(* IEC 61131-3 sources: SRCI/RobotLibrary/Library/POUs/BasicMove/MC_ReturnToPrimary, 1 file *)

(* ---- MC_ReturnToPrimaryFB.st ---- *)
/// Return to path left during active interrupt
FUNCTION_BLOCK MC_ReturnToPrimaryFB EXTENDS RobotLibraryBaseFB
// -------------------------------------------------------------------------
//  SRCI Robot Library
// -------------------------------------------------------------------------
//
//  Object:      ReturnToPrimaryFB
//  Author:      Thorsten Brach
//  Date:        2024-06-01
//
//  Description:
//
//
//  Copyright:
//    (C) 2024 Thorsten Brach. All rights reserved
//             Licensed under the LGPL-3.0 license.
//
//  Disclaimer:
//    This project is provided without any guarantee and can be used for
//    private and commercial purposes. Any use is at the user’s
//    own risk and responsibility.
//
// -------------------------------------------------------------------------
VAR_INPUT
  /// Activate ReturnToPrimary
  Enable             : BOOL;
  /// command parameter
  ParCmd             : ReturnToPrimaryParCmd;
END_VAR

VAR_OUTPUT
  /// The command has been completed successfully
  Done               : BOOL;
  /// FB is being processed
  Busy               : BOOL;
  /// Command is transferred and confirmed by the RC
  CommandBuffered    : BOOL;
  /// The command takes control of the motion of the according axis group
  Active             : BOOL;
  /// The command was aborted by another command.
  CommandAborted     : BOOL;
  /// TRUE, while command is interrupted during execution and can be continued
  CommandInterrupted : BOOL;
  /// command results
  OutCmd             : ReturnToPrimaryOutCmd;
END_VAR

VAR
  /// internal copy of command parameter
 _parCmd             : ReturnToPrimaryParCmd;
  /// command data to send
 _command            : ReturnToPrimarySendData;
  /// response data received
 _response           : ReturnToPrimaryRecvData;
  /// Rising edge for enable
 _enable_R           : R_TRIG;
  /// Falling edge for enable
 _enable_F           : F_TRIG;
END_VAR

  SUPER^(AxesGroup := AxesGroup);

END_FUNCTION_BLOCK

METHOD INTERNAL CheckAddParameter : BOOL
VAR_INPUT
  /// Payload pointer
  PayloadPtr : UDINT;
END_VAR
VAR
  /// Payload as byte array
  Payload    : ARRAY [1..SIZEOF(_command)] OF BYTE;
  /// Null Byte array
  Null       : ARRAY [1..SIZEOF(_command)] OF BYTE;
  /// Data length to compare
  DataLen    : UDINT;
END_VAR

  // Payload pointer must be decreased by one byte, because ADR(Payload) is already one byte !
  PayloadPtr := LIMIT (0, PayloadPtr - 1, SIZEOF(Payload) -1);
  // Convert command struct to payload array
  SysDepMemCpy( pDest := ADR(Payload), pSrc := ADR(_command), DataLen := SIZEOF(_command));
  // Calculate the data length to compare - at least one byte must be compared !
  DataLen := LIMIT(1, SIZEOF(Payload) - PayloadPtr, SIZEOF(Payload));
  // Compare Payload-Array with Null-Byte-Array
  CheckAddParameter := SysDepMemCmp( pData1 := ADR(Payload) + PayloadPtr , pData2 := ADR(Null), DataLen := DataLen) <>  RobotLibraryConstants.OK ;

END_METHOD

METHOD PROTECTED CheckFunctionSupported : BOOL
VAR_IN_OUT
  /// Robot assignment of function
  AxesGroup : AxesGroup;
END_VAR

  CheckFunctionSupported := AxesGroup.State.RobotData.RCSupportedFunctions.ReturnToPrimary;

  IF ( NOT CheckFunctionSupported )
  THEN
    // call base implementation for set error and create log entry
    SUPER^.CheckFunctionSupported(AxesGroup := AxesGroup);
  END_IF

END_METHOD

METHOD PROTECTED CheckParameterChanged : BOOL
VAR_IN_OUT
  /// Robot assignment of function
  AxesGroup    : AxesGroup;
END_VAR

  // Check ParCmd Size is > 0, because MemCmp does not work correctly with size = 0
  IF (SIZEOF(ParCmd) = 0) OR (_stepCmd = 0)
  THEN
    RETURN;
  END_IF

  // compare memory
  _parameterChanged := ( SysDepMemCmp(pData1 := ADR(ParCmd), pData2 := ADR(_parCmd), DataLen := SIZEOF(ParCmd)) <> RobotLibraryConstants.OK );

  // check parameter valid ?
  _parameterValid   := CheckParameterValid( AxesGroup := AxesGroup );

  IF ((  _parameterChanged        )  AND
      (  _parameterValid          )) OR
      (  _parameterUpdateInternal )
  THEN
    // reset internal flag for send parameter update
   _parameterUpdateInternal := FALSE;
    // update internal copy of parameters
   _parCmd := ParCmd;
    // inc parameter sequence
   _command.ParSeq := _command.ParSeq + 1;
    // update command data
    CommandData := CreateCommandPayload(AxesGroup := AxesGroup); // ( Access via reference to rCommandFB in ACR )
    // notify active command register
    AxesGroup.Acyclic.ActiveCommandRegister.NotifyParameterChanged := _uniqueID;
  END_IF

END_METHOD

METHOD PROTECTED CheckParameterValid : BOOL
VAR_IN_OUT
  /// Robot assignment of function
  AxesGroup : AxesGroup;
END_VAR
VAR
  /// internal index for loops
 _idx : DINT;
END_VAR

  CheckParameterValid := TRUE;

  // Check ParCmd.ReturnMode valid ?
  IF (( ParCmd.ReturnMode <> ReturnMode.INTERRUPT_POSITION ) AND
      ( ParCmd.ReturnMode <> ReturnMode.END_POSITION       ))
  THEN
    // Parameter not valid
    CheckParameterValid := FALSE;
    // Set error
    ErrorID := RobotLibraryErrorIdEnum.ERR_INVALID_PAR_CMD;
    // Create log entry
    CreateLogMessagePara1 ( Timestamp   := AxesGroup.State.SystemTime,
                            MessageType := MessageType.CMD,
                            Severity    := Severity.ERROR,
                            MessageCode := ErrorID,
                            MessageText := 'Invalid Parameter ParCmd.ReturnMode = {1}',
                            Para1       := RETURN_MODE_TO_STRING(ParCmd.ReturnMode));
    RETURN;
  END_IF

  // Check ParCmd.VelocityRate valid ?
  IF  (( SysDepIsValidReal(ParCmd.VelocityRate) = FALSE )  OR
      ((                   ParCmd.VelocityRate  <     0 )  AND
       (                   ParCmd.VelocityRate <>    -1 )) OR
       (                   ParCmd.VelocityRate  >   100 ))
  THEN
    // Parameter not valid
    CheckParameterValid := FALSE;
    // Set error
    ErrorID := RobotLibraryErrorIdEnum.ERR_VELOCITY_INVALID;
    // Create log entry
    CreateLogMessagePara1 ( Timestamp   := AxesGroup.State.SystemTime,
                            MessageType := MessageType.CMD,
                            Severity    := Severity.ERROR,
                            MessageCode := ErrorID,
                            MessageText := 'Invalid Parameter ParCmd.VelocityRate = {1}',
                            Para1       := VALID_REAL_TO_STRING(ParCmd.VelocityRate));
    RETURN;
  END_IF

  // Check ParCmd.AccelerationRate valid ?
  IF  (( SysDepIsValidReal(ParCmd.AccelerationRate) = FALSE )  OR
      ((                   ParCmd.AccelerationRate  <     0 )  AND
       (                   ParCmd.AccelerationRate <>    -1 )) OR
       (                   ParCmd.AccelerationRate  >   100 ))
  THEN
    // Parameter not valid
    CheckParameterValid := FALSE;
    // Set error
    ErrorID := RobotLibraryErrorIdEnum.ERR_ACCELERATION_INVALID;
    // Create log entry
    CreateLogMessagePara1 ( Timestamp   := AxesGroup.State.SystemTime,
                            MessageType := MessageType.CMD,
                            Severity    := Severity.ERROR,
                            MessageCode := ErrorID,
                            MessageText := 'Invalid Parameter ParCmd.AccelerationRate = {1}',
                            Para1       := VALID_REAL_TO_STRING(ParCmd.AccelerationRate));
    RETURN;
  END_IF

  // Check ParCmd.DecelerationRate valid ?
  IF  (( SysDepIsValidReal(ParCmd.DecelerationRate) = FALSE )  OR
      ((                   ParCmd.DecelerationRate  <     0 )  AND
       (                   ParCmd.DecelerationRate <>    -1 )) OR
       (                   ParCmd.DecelerationRate  >   100 ))
  THEN
    // Parameter not valid
    CheckParameterValid := FALSE;
    // Set error
    ErrorID := RobotLibraryErrorIdEnum.ERR_DECELERATION_INVALID;
    // Create log entry
    CreateLogMessagePara1 ( Timestamp   := AxesGroup.State.SystemTime,
                            MessageType := MessageType.CMD,
                            Severity    := Severity.ERROR,
                            MessageCode := ErrorID,
                            MessageText := 'Invalid Parameter ParCmd.DecelerationRate = {1}',
                            Para1       := VALID_REAL_TO_STRING(ParCmd.DecelerationRate));
    RETURN;
  END_IF

  // Check ParCmd.JerkRate valid ?
  IF  (( SysDepIsValidReal(ParCmd.JerkRate) = FALSE )  OR
      ((                   ParCmd.JerkRate  <     0 )  AND
       (                   ParCmd.JerkRate <>    -1 )) OR
       (                   ParCmd.JerkRate  >   100 ))
  THEN
    // Parameter not valid
    CheckParameterValid := FALSE;
    // Set error
    ErrorID := RobotLibraryErrorIdEnum.ERR_JERK_INVALID;
    // Create log entry
    CreateLogMessagePara1 ( Timestamp   := AxesGroup.State.SystemTime,
                            MessageType := MessageType.CMD,
                            Severity    := Severity.ERROR,
                            MessageCode := ErrorID,
                            MessageText := 'Invalid Parameter ParCmd.JerkRate = {1}',
                            Para1       := VALID_REAL_TO_STRING(ParCmd.JerkRate));
    RETURN;
  END_IF

  // Check ParCmd.ToolNo valid ?
  IF (( ParCmd.ToolNo <   0                                                ) OR
      ( ParCmd.ToolNo > 254                                                ) OR
      ( ParCmd.ToolNo > AxesGroup.State.ConfigurationData.HighestToolIndex ) OR
      ( ParCmd.ToolNo > RobotLibraryParameter.TOOL_MAX -1                  ))
  THEN
    // Parameter not valid
    CheckParameterValid := FALSE;

    // Check ToolNo available on RC ?
    IF ( ParCmd.ToolNo > AxesGroup.State.ConfigurationData.HighestToolIndex )
    THEN
      ErrorID := RobotLibraryErrorIdEnum.ERR_TOOLNO_UNAVAILABLE;
    ELSE
      ErrorID := RobotLibraryErrorIdEnum.ERR_TOOLNO_RANGE;
  	END_IF

    // Create log entry
    CreateLogMessagePara1 ( Timestamp   := AxesGroup.State.SystemTime,
                            MessageType := MessageType.CMD,
                            Severity    := Severity.ERROR,
                            MessageCode := ErrorID,
                            MessageText := 'Invalid Parameter ParCmd.ToolNo = {1}',
                            Para1       := USINT_TO_STRING(ParCmd.ToolNo));
    RETURN;
  END_IF

  // Check ParCmd.FrameNo valid ?
  IF (( ParCmd.FrameNo <   0                                                 ) OR
      ( ParCmd.FrameNo > 254                                                 ) OR
      ( ParCmd.FrameNo > AxesGroup.State.ConfigurationData.HighestFrameIndex ) OR
      ( ParCmd.FrameNo > RobotLibraryParameter.FRAME_MAX -1                  ))
  THEN
    // Parameter not valid
    CheckParameterValid := FALSE;

    // Check FrameNo available on RC ?
    IF ( ParCmd.FrameNo > AxesGroup.State.ConfigurationData.HighestFrameIndex )
    THEN
      ErrorID := RobotLibraryErrorIdEnum.ERR_FRAMENO_UNAVAILABLE;
    ELSE
      ErrorID := RobotLibraryErrorIdEnum.ERR_FRAMENO_RANGE;
  	END_IF

    // Create log entry
    CreateLogMessagePara1 ( Timestamp   := AxesGroup.State.SystemTime,
                            MessageType := MessageType.CMD,
                            Severity    := Severity.ERROR,
                            MessageCode := ErrorID,
                            MessageText := 'Invalid Parameter ParCmd.FrameNo = {1}',
                            Para1       := USINT_TO_STRING(ParCmd.FrameNo));
    RETURN;
  END_IF

  // Check ParCmd.DistanceLimit valid ?
  IF  ( SysDepIsValidReal(ParCmd.DistanceLimit) = FALSE )
  THEN
    // Parameter not valid
    CheckParameterValid := FALSE;
    // Set error
    ErrorID := RobotLibraryErrorIdEnum.ERR_JERK_INVALID;
    // Create log entry
    CreateLogMessagePara1 ( Timestamp   := AxesGroup.State.SystemTime,
                            MessageType := MessageType.CMD,
                            Severity    := Severity.ERROR,
                            MessageCode := ErrorID,
                            MessageText := 'Invalid Parameter ParCmd.DistanceLimit = {1}',
                            Para1       := VALID_REAL_TO_STRING(ParCmd.DistanceLimit));
    RETURN;
  END_IF

  // Check ParCmd.TrajectoryMode valid ?
  IF (( ParCmd.TrajectoryMode <> TrajectoryMode.INVALID         ) AND
      ( ParCmd.TrajectoryMode <> TrajectoryMode.LINEAR_MOVEMENT ) AND
      ( ParCmd.TrajectoryMode <> TrajectoryMode.PTP_MOVEMENT    ))
  THEN
    // Parameter not valid
    CheckParameterValid := FALSE;
    // Set error
    ErrorID := RobotLibraryErrorIdEnum.ERR_TRAJECTORYMODE_INVALID;
    // Create log entry
    CreateLogMessagePara1 ( Timestamp   := AxesGroup.State.SystemTime,
                            MessageType := MessageType.CMD,
                            Severity    := Severity.ERROR,
                            MessageCode := ErrorID,
                            MessageText := 'Invalid Parameter ParCmd.TrajectoryMode = {1}',
                            Para1       := TRAJECTORY_MODE_TO_STRING(ParCmd.TrajectoryMode));
    RETURN;
  END_IF

  // Check ParCmd.MoveTime valid ?
  IF  ( ParCmd.MoveTime < T#0S )
  THEN
    // Parameter not valid
    CheckParameterValid := FALSE;
    // Set error
    ErrorID := RobotLibraryErrorIdEnum.ERR_INVALID_PAR_CMD;
    // Create log entry
    CreateLogMessagePara1 ( Timestamp   := AxesGroup.State.SystemTime,
                            MessageType := MessageType.CMD,
                            Severity    := Severity.ERROR,
                            MessageCode := ErrorID,
                            MessageText := 'Invalid Parameter ParCmd.MoveTime = {1}',
                            Para1       := TIME_TO_STRING(ParCmd.MoveTime));
    RETURN;
  END_IF

  // Check ParCmd.AllowDifferences
  // -> no plausibility check for boolean

END_METHOD

METHOD INTERNAL CreateCommandPayload : RobotLibraryCommandDataFB
VAR_IN_OUT
  /// Robot assignment of function
  AxesGroup : AxesGroup;
END_VAR
VAR
  /// Parameter count
 _parameterCnt : DINT;
END_VAR
// Table 6-310: Sent CMD payload (PLC to RC) of "ReturnToPrimary"
// --------------------------
// Header
// --------------------------
// Byte 00 : UINT  - Type HB
// Byte 01 :       - Type LB
// Byte 02 : USINT - Reserve | ExecutionMode
// Byte 03 : USINT - ParSeq  | Priority
// --------------------------
// Datablock
// --------------------------
// Byte 04  : UINT  - VelocityRate LW HB
// Byte 05  :       - VelocityRate LW LB
// Byte 06  : UINT  - AccelerationRate LW HB
// Byte 07  :       - AccelerationRate LW LB
// Byte 08  : UINT  - DecelerationRate LW HB
// Byte 09  :       - DecelerationRate LW LB
// Byte 10  : UINT  - JerkRate LW HB
// Byte 11  :       - JerkRate LW LB
// Byte 12  : REAL  - DistanceLimit HW HB
// Byte 13  :       - DistanceLimit HW LB
// Byte 14  :       - DistanceLimit LW HB
// Byte 15  :       - DistanceLimit LW LB
// Byte 16  : USINT - ToolNo
// Byte 17  : USINT - FrameNo
// Byte 18  : UINT  - Move Time LW HB
// Byte 19  : UINT  - Move Time LW LB
// Byte 20  : BYTE  - BIT 00 : ReturnMode
//                    BIT 01 : TrajectoryMode
//                    BIT 02 : Enable
//                    BIT 03 : AllowDifferences
// Byte 21  : BYTE  - PaddingByte

// --------------------------
VAR
 _tmpByte : BYTE;
END_VAR

  // set command parameter
  _command.CmdTyp            :=  CmdType.ReturnToPrimary;
  _command.ExecMode          :=  ExecMode;
  _command.ParSeq            := _command.ParSeq;
  _command.Priority          :=  Priority;
  _command.ToolNo            := _parCmd.ToolNo;
  _command.FrameNo           := _parCmd.FrameNo;
  _command.VelocityRate      :=  REAL_TO_PERCENT_UINT(_parCmd.VelocityRate     , IsOptional := FALSE);
  _command.AccelerationRate  :=  REAL_TO_PERCENT_UINT(_parCmd.AccelerationRate , IsOptional := FALSE);
  _command.DecelerationRate  :=  REAL_TO_PERCENT_UINT(_parCmd.DecelerationRate , IsOptional := TRUE );
  _command.JerkRate          :=  REAL_TO_PERCENT_UINT(_parCmd.JerkRate         , IsOptional := TRUE );
  _command.DistanceLimit     := _parCmd.DistanceLimit;
  _command.ReturnMode        :=(_parCmd.ReturnMode = ReturnMode.END_POSITION);
  _command.TrajectoryMode    := _parCmd.TrajectoryMode = TrajectoryMode.PTP_MOVEMENT;
  _command.MoveTime          :=  TIME_TO_UINT(_parCmd.MoveTime);
  _command.Enable            :=  Enable;

  // copy command data to header
  _cmdHeader := _command;
  // call base implementation to copy header to payload buffer
  CreateCommandPayload := SUPER^.CreateCommandPayload(AxesGroup := AxesGroup);

  {warning 'ToDo: Changes in Spec V1.5, which are different to Spec V1.3'}

  // Check parameter must be added ?
  IF ( CheckAddParameter(CreateCommandPayload.PayloadPtr))
  THEN
    // add command.VelocityRate
    CreateCommandPayload.AddUint(_command.VelocityRate);
    // inc parameter counter
   _parameterCnt := _parameterCnt + 1;
  END_IF

  // Check parameter must be added ?
  IF ( CheckAddParameter(CreateCommandPayload.PayloadPtr))
  THEN
    // add command.AccelerationRate
    CreateCommandPayload.AddUint(_command.AccelerationRate);
    // inc parameter counter
   _parameterCnt := _parameterCnt + 1;
  END_IF

  // Check parameter must be added ?
  IF ( CheckAddParameter(CreateCommandPayload.PayloadPtr))
  THEN
    // add command.DecelerationRate
    CreateCommandPayload.AddUint(_command.DecelerationRate);
    // inc parameter counter
   _parameterCnt := _parameterCnt + 1;
  END_IF

  // Check parameter must be added ?
  IF ( CheckAddParameter(CreateCommandPayload.PayloadPtr))
  THEN
    // add command.JerkRate
    CreateCommandPayload.AddUint(_command.JerkRate);
    // inc parameter counter
   _parameterCnt := _parameterCnt + 1;
  END_IF

  // Check parameter must be added ?
  IF ( CheckAddParameter(CreateCommandPayload.PayloadPtr))
  THEN
    // add command.DistanceLimit
    CreateCommandPayload.AddReal(_command.DistanceLimit);
    // inc parameter counter
   _parameterCnt := _parameterCnt + 1;
  END_IF

  // Check parameter must be added ?
  IF ( CheckAddParameter(CreateCommandPayload.PayloadPtr))
  THEN
    // add command.ToolNo
    CreateCommandPayload.AddUsint(_command.ToolNo);
    // inc parameter counter
   _parameterCnt := _parameterCnt + 1;
  END_IF

  // Check parameter must be added ?
  IF ( CheckAddParameter(CreateCommandPayload.PayloadPtr))
  THEN
    // add command.FrameNo
    CreateCommandPayload.AddUsint(_command.FrameNo);
    // inc parameter counter
   _parameterCnt := _parameterCnt + 1;
  END_IF

  // Check parameter must be added ?
  IF ( CheckAddParameter(CreateCommandPayload.PayloadPtr))
  THEN
    // add command.MoveTime
    CreateCommandPayload.AddUint(_command.MoveTime);
    // inc parameter counter
   _parameterCnt := _parameterCnt + 1;
  END_IF

  // Check parameter must be added ?
  IF ( CheckAddParameter(CreateCommandPayload.PayloadPtr))
  THEN
   _tmpByte.0 := _command.ReturnMode;
   _tmpByte.1 := _command.TrajectoryMode;
   _tmpByte.2 := _command.Enable;
   _tmpByte.3 := _command.AllowDifferences;
    // add command.ReturnMode
    CreateCommandPayload.AddByte(_tmpByte);
    // inc parameter counter
   _parameterCnt := _parameterCnt + 1;
  END_IF

  // Create logging
  CreateCommandPayloadLog(AxesGroup := AxesGroup, ParameterCnt := _parameterCnt);

END_METHOD

METHOD INTERNAL CreateCommandPayloadLog
VAR_IN_OUT
  /// Robot assignment of function
  AxesGroup : AxesGroup;
END_VAR
VAR_INPUT
  /// Parameter count
  ParameterCnt : DINT;
END_VAR

  // Create log entry for Parameter start
  CreateLogMessagePara1 ( Timestamp   := AxesGroup.State.SystemTime,
                          MessageType := MessageType.CMD,
                          Severity    := Severity.DEBUG,
                          MessageCode := 0,
                          MessageText := 'Create command payload with the {1} parameter(s) :',
                          Para1       := DINT_TO_STRING(ParameterCnt));

  // Return if no parameter is remaining...
  IF ( ParameterCnt = 0 ) THEN RETURN; END_IF
  // dec remaining parameter(s)
  ParameterCnt := ParameterCnt - 1;
  // Create log entry for ToolNo
  CreateLogMessagePara1 ( Timestamp   := AxesGroup.State.SystemTime,
                          MessageType := MessageType.CMD,
                          Severity    := Severity.DEBUG,
                          MessageCode := 0,
                          MessageText := 'Command.ToolNo = {1}',
                          Para1       :=  USINT_TO_STRING(_command.ToolNo));

  // Return if no parameter is remaining...
  IF ( ParameterCnt = 0 ) THEN RETURN; END_IF
  // dec remaining parameter(s)
  ParameterCnt := ParameterCnt - 1;
  // Create log entry for FrameNo
  CreateLogMessagePara1 ( Timestamp   := AxesGroup.State.SystemTime,
                          MessageType := MessageType.CMD,
                          Severity    := Severity.DEBUG,
                          MessageCode := 0,
                          MessageText := 'Command.FrameNo = {1}',
                          Para1       :=  USINT_TO_STRING(_command.FrameNo));

  // Return if no parameter is remaining...
  IF ( ParameterCnt = 0 ) THEN RETURN; END_IF
  // dec remaining parameter(s)
  ParameterCnt := ParameterCnt - 1;
  // Create log entry for VelocityRate
  CreateLogMessagePara1 ( Timestamp   := AxesGroup.State.SystemTime,
                          MessageType := MessageType.CMD,
                          Severity    := Severity.DEBUG,
                          MessageCode := 0,
                          MessageText := 'Command.VelocityRate = {1}',
                          Para1       :=  UINT_TO_STRING(_command.VelocityRate));

  // Return if no parameter is remaining...
  IF ( ParameterCnt = 0 ) THEN RETURN; END_IF
  // dec remaining parameter(s)
  ParameterCnt := ParameterCnt - 1;
  // Create log entry for AccelerationRate
  CreateLogMessagePara1 ( Timestamp   := AxesGroup.State.SystemTime,
                          MessageType := MessageType.CMD,
                          Severity    := Severity.DEBUG,
                          MessageCode := 0,
                          MessageText := 'Command.AccelerationRate = {1}',
                          Para1       :=  UINT_TO_STRING(_command.AccelerationRate));

  // Return if no parameter is remaining...
  IF ( ParameterCnt = 0 ) THEN RETURN; END_IF
  // dec remaining parameter(s)
  ParameterCnt := ParameterCnt - 1;
  // Create log entry for DecelerationRate
  CreateLogMessagePara1 ( Timestamp   := AxesGroup.State.SystemTime,
                          MessageType := MessageType.CMD,
                          Severity    := Severity.DEBUG,
                          MessageCode := 0,
                          MessageText := 'Command.DecelerationRate = {1}',
                          Para1       :=  UINT_TO_STRING(_command.DecelerationRate));

  // Return if no parameter is remaining...
  IF ( ParameterCnt = 0 ) THEN RETURN; END_IF
  // dec remaining parameter(s)
  ParameterCnt := ParameterCnt - 1;
  // Create log entry for JerkRate
  CreateLogMessagePara1 ( Timestamp   := AxesGroup.State.SystemTime,
                          MessageType := MessageType.CMD,
                          Severity    := Severity.DEBUG,
                          MessageCode := 0,
                          MessageText := 'Command.JerkRate = {1}',
                          Para1       :=  UINT_TO_STRING(_command.JerkRate));

  // Return if no parameter is remaining...
  IF ( ParameterCnt = 0 ) THEN RETURN; END_IF
  // dec remaining parameter(s)
  ParameterCnt := ParameterCnt - 1;
  // Create log entry for DistanceLimit
  CreateLogMessagePara1 ( Timestamp   := AxesGroup.State.SystemTime,
                          MessageType := MessageType.CMD,
                          Severity    := Severity.DEBUG,
                          MessageCode := 0,
                          MessageText := 'Command.DistanceLimit = {1}',
                          Para1       :=  REAL_TO_STRING(_command.DistanceLimit));

  // Return if no parameter is remaining...
  IF ( ParameterCnt = 0 ) THEN RETURN; END_IF
  // dec remaining parameter(s)
  ParameterCnt := ParameterCnt - 1;
  // Create log entry for ReturnMode
  CreateLogMessagePara1 ( Timestamp   := AxesGroup.State.SystemTime,
                          MessageType := MessageType.CMD,
                          Severity    := Severity.DEBUG,
                          MessageCode := 0,
                          MessageText := 'Command.ReturnMode = {1}',
                          Para1       :=  BOOL_TO_STRING(_command.ReturnMode));

  // Return if no parameter is remaining...
  IF ( ParameterCnt = 0 ) THEN RETURN; END_IF
  // dec remaining parameter(s)
  ParameterCnt := ParameterCnt - 1;
  // Create log entry for TrajectoryMode
  CreateLogMessagePara1 ( Timestamp   := AxesGroup.State.SystemTime,
                          MessageType := MessageType.CMD,
                          Severity    := Severity.DEBUG,
                          MessageCode := 0,
                          MessageText := 'Command.TrajectoryMode = {1}',
                          Para1       :=  BOOL_TO_STRING(_command.TrajectoryMode));

  // Return if no parameter is remaining...
  IF ( ParameterCnt = 0 ) THEN RETURN; END_IF
  // dec remaining parameter(s)
  ParameterCnt := ParameterCnt - 1;
  // Create log entry for MoveTime
  CreateLogMessagePara1 ( Timestamp   := AxesGroup.State.SystemTime,
                          MessageType := MessageType.CMD,
                          Severity    := Severity.DEBUG,
                          MessageCode := 0,
                          MessageText := 'Command.MoveTime = {1}',
                          Para1       :=  UINT_TO_STRING(_command.MoveTime));

END_METHOD

METHOD FB_init : BOOL
VAR_INPUT
  /// if TRUE, the retain variables are initialized (warm start / cold start)
  bInitRetains : BOOL;
  /// if TRUE, the instance afterwards gets moved into the copy code (online change)
  bInCopyCode  : BOOL;
END_VAR

  MyType := 'MC_ReturnToPrimaryFB';

  ExecMode := ExecutionMode.SEQUENCE_PRIMARY;
  Priority := PriorityLevel.NORMAL;

END_METHOD

METHOD PROTECTED OnExecRun : DINT
VAR_IN_OUT
  /// Robot assignment of function
  AxesGroup : AxesGroup;
END_VAR

  // call base implementation
  SUPER^.OnExecRun(AxesGroup := AxesGroup);

  // building rising and falling edges
  _enable_R( CLK := Enable);
  _enable_F( CLK := Enable);

  CASE _stepCmd OF

    00:  IF ( _enable_R.Q ) AND ( NOT Error)
         THEN
           // reset the rising edge
          _enable_R();
           // reset the falling edge
          _enable_F();

           // Check function is supported and parameter are valid ?
           IF (( CheckFunctionSupported( AxesGroup := AxesGroup )) AND
               ( CheckParameterValid   ( AxesGroup := AxesGroup )))
           THEN
             // set busy flag
             Busy := TRUE;
             // Reset command outputs
             SysDepMemSet(pDest := ADR(OutCmd), Value := 0, DataLen := SIZEOF(OutCmd));
             // apply command parameter
            _parCmd := ParCmd;
             // init parameter sequence
            _command.ParSeq := 1;
             // create command data
             CommandData := CreateCommandPayload(AxesGroup := AxesGroup);
             // Add command to active command register
            _uniqueID := AxesGroup.Acyclic.ActiveCommandRegister.AddCmd( pCommandFB := ADR(THIS^ ));
             // set timeout
             SetTimeout(PT := _timeoutCmd, rTimer := _timerCmd);
             // inc step counter
            _stepCmd := _stepCmd + 1;
           END_IF
         END_IF

    01:  // Wait for responce received
         IF ( _responseReceived )
         THEN
           // reset response received flag
          _responseReceived := FALSE;
           // reset Active flag
           Active := FALSE;

           CASE  _response.State
           OF
             CmdMessageState.BUFFERED    : CommandBuffered    := TRUE;
             CmdMessageState.ACTIVE      : Active             := TRUE;
             CmdMessageState.INTERRUPTED : CommandInterrupted := TRUE;
             CmdMessageState.DONE        : Done               := TRUE;
             CmdMessageState.ABORTED     : CommandAborted     := TRUE;
             CmdMessageState.ERROR       : Error              := TRUE;
           END_CASE

           // Done, Aborted or Error ?
           IF (_response.State >= CmdMessageState.DONE )
           THEN
             // Reset Busy flag
             Busy := FALSE;
             // Update results
             OutCmd.Progress          :=  PERCENT_UINT_TO_REAL( Value := _response.Progress, IsOptional := FALSE);
             OutCmd.RemainingDistance := _response.RemainingDistance;
             OutCmd.PrimaryPosToolNo  := UINT_TO_USINT(_response.PrimaryPosToolNo);  {warning 'ToDo'}
             OutCmd.PrimaryPosFrameNo := UINT_TO_USINT(_response.PrimaryPosFrameNo); {warning 'ToDo'}

             // set timeout
             SetTimeout(PT := _timeoutCmd, rTimer := _timerCmd);
             // inc step counter
            _stepCmd := _stepCmd + 1;
           END_IF
         END_IF

    02: IF (NOT Enable)
        THEN
          Reset();
        END_IF

  ELSE
    // invalid step
    ErrorID := RobotLibraryErrorIdEnum.ERR_INVALID_STEP;
  END_CASE

  // Reset FB
  IF (( _enable_R.Q ) OR
      ( _enable_F.Q ))
  THEN
    Reset();
  END_IF

END_METHOD

METHOD INTERNAL ParseResponsePayload : DINT
VAR_INPUT
  /// Response data
  ResponseData : RobotLibraryResponseDataFB;
  /// Timestamp
  Timestamp    : SystemTime;
END_VAR
VAR
  /// Parameter count
 _parameterCnt : DINT;
END_VAR
// Table 6-311: Received CMD payload (RC to PLC) of "ReturnToPrimary"
// --------------------------
// Header
// --------------------------
// Byte 00 : USINT - ParSeq | State
// Byte 01 : SINT  - AlarmMessageSeverity
// Byte 02 : UINT  - AlarmMessageCode HB
// Byte 03 :       - AlarmMessageCode LB
// --------------------------
// Datablock
// --------------------------
// Byte 04 : UINT  - Progress LW HB
// Byte 05 :       - Progress LW LB
// Byte 06 : REAL  - RemainingDistance HW HB
// Byte 07 :       - RemainingDistance HW LB
// Byte 08 :       - RemainingDistance LW HB
// Byte 09 :       - RemainingDistance LW LB
// Byte 10 : USINT - PrimaryPosToolNo
// Byte 11 : USINT - PrimaryPosToolNo
// --------------------------

  // call base implementation to parse the header from payload buffer
  ResponseData.PayloadPtr := SUPER^.ParseResponsePayload(ResponseData := ResponseData, Timestamp := Timestamp);

  // copy parsed header to response
  _response.ParSeq               := _rspHeader.ParSeq;
  _response.State                := _rspHeader.State;
  _response.AlarmMessageSeverity := _rspHeader.AlarmMessageSeverity;
  _response.AlarmMessageCode     := _rspHeader.AlarmMessageCode;

  // Check payload remaining ?
  IF ( ResponseData.IsPayloadRemaining)
  THEN
    // Get Response.Progress
   _response.Progress             := ResponseData.GetUint();
    // inc parameter counter
   _parameterCnt := _parameterCnt + 1;
  END_IF

  // Check payload remaining ?
  IF ( ResponseData.IsPayloadRemaining)
  THEN
    // Get Response.RemainingDistance
   _response.RemainingDistance    := ResponseData.GetReal();
    // inc parameter counter
   _parameterCnt := _parameterCnt + 1;
  END_IF

  // Check payload remaining ?
  IF ( ResponseData.IsPayloadRemaining)
  THEN
    // Get Response.PrimaryPosToolNo
   _response.PrimaryPosToolNo     := ResponseData.GetUsint();
    // inc parameter counter
   _parameterCnt := _parameterCnt + 1;
  END_IF

  // Check payload remaining ?
  IF ( ResponseData.IsPayloadRemaining)
  THEN
    // Get Response.PrimaryPosFrameNo
   _response.PrimaryPosFrameNo    := ResponseData.GetUsint();
    // inc parameter counter
   _parameterCnt := _parameterCnt + 1;
  END_IF

  // Create logging
  ParseResponsePayloadLog(ResponseData := ResponseData, Timestamp := Timestamp, ParameterCnt := _parameterCnt);

END_METHOD

METHOD INTERNAL ParseResponsePayloadLog
VAR_INPUT
  /// Response data
  ResponseData : RobotLibraryResponseDataFB;
  /// Timestamp
  Timestamp    : SystemTime;
  /// Parameter count
  ParameterCnt : DINT;
END_VAR

  // Create log entry for Parameter start
  CreateLogMessagePara1 ( Timestamp   := Timestamp,
                          MessageType := MessageType.CMD,
                          Severity    := Severity.DEBUG,
                          MessageCode := 0,
                          MessageText := '{1} parameter(s) to parse from the response data:',
                          Para1       := DINT_TO_STRING(ParameterCnt));

  // Return if no parameter is remaining...
  IF ( ParameterCnt = 0 ) THEN RETURN; END_IF
  // dec remaining parameter(s)
  ParameterCnt := ParameterCnt - 1;
  // Create log entry for Progress
  CreateLogMessagePara1 ( Timestamp   := Timestamp,
                          MessageType := MessageType.CMD,
                          Severity    := Severity.DEBUG,
                          MessageCode := 0,
                          MessageText := 'Response.Progress = {1}',
                          Para1       :=  UINT_TO_STRING(_response.Progress));

  // Return if no parameter is remaining...
  IF ( ParameterCnt = 0 ) THEN RETURN; END_IF
  // dec remaining parameter(s)
  ParameterCnt := ParameterCnt - 1;
  // Create log entry for RemainingDistance
  CreateLogMessagePara1 ( Timestamp   := Timestamp,
                          MessageType := MessageType.CMD,
                          Severity    := Severity.DEBUG,
                          MessageCode := 0,
                          MessageText := 'Response.RemainingDistance = {1}',
                          Para1       :=  REAL_TO_STRING(_response.RemainingDistance));

  // Return if no parameter is remaining...
  IF ( ParameterCnt = 0 ) THEN RETURN; END_IF
  // dec remaining parameter(s)
  ParameterCnt := ParameterCnt - 1;
  // Create log entry for PrimaryPosToolNo
  CreateLogMessagePara1 ( Timestamp   := Timestamp,
                          MessageType := MessageType.CMD,
                          Severity    := Severity.DEBUG,
                          MessageCode := 0,
                          MessageText := 'Response.PrimaryPosToolNo = {1}',
                          Para1       :=  UINT_TO_STRING(_response.PrimaryPosToolNo));

  // Return if no parameter is remaining...
  IF ( ParameterCnt = 0 ) THEN RETURN; END_IF
  // dec remaining parameter(s)
  ParameterCnt := ParameterCnt - 1;
  // Create log entry for PrimaryPosFrameNo
  CreateLogMessagePara1 ( Timestamp   := Timestamp,
                          MessageType := MessageType.CMD,
                          Severity    := Severity.DEBUG,
                          MessageCode := 0,
                          MessageText := 'Response.PrimaryPosFrameNo = {1}',
                          Para1       :=  UINT_TO_STRING(_response.PrimaryPosFrameNo));

END_METHOD

METHOD PROTECTED Reset : DINT
VAR_INPUT
END_VAR

  Reset := SUPER^.Reset();

  Done               := FALSE;
  Busy               := FALSE;
  Active             := FALSE;
  CommandBuffered    := FALSE;
  CommandAborted     := FALSE;
  CommandInterrupted := FALSE;

END_METHOD
